(* PLC project Unnamed, Unknown Unnamed 1 *)
(* stored: creationDateTime 2022-08-16T15:49:17, modificationDateTime 2023-01-11T10:21:23 *)

PROGRAM Blink
  VAR
    blink_led AT %QX0.5 : BOOL;
  END_VAR
  VAR
    TON0 : TON;
    TOF0 : TOF;
  END_VAR

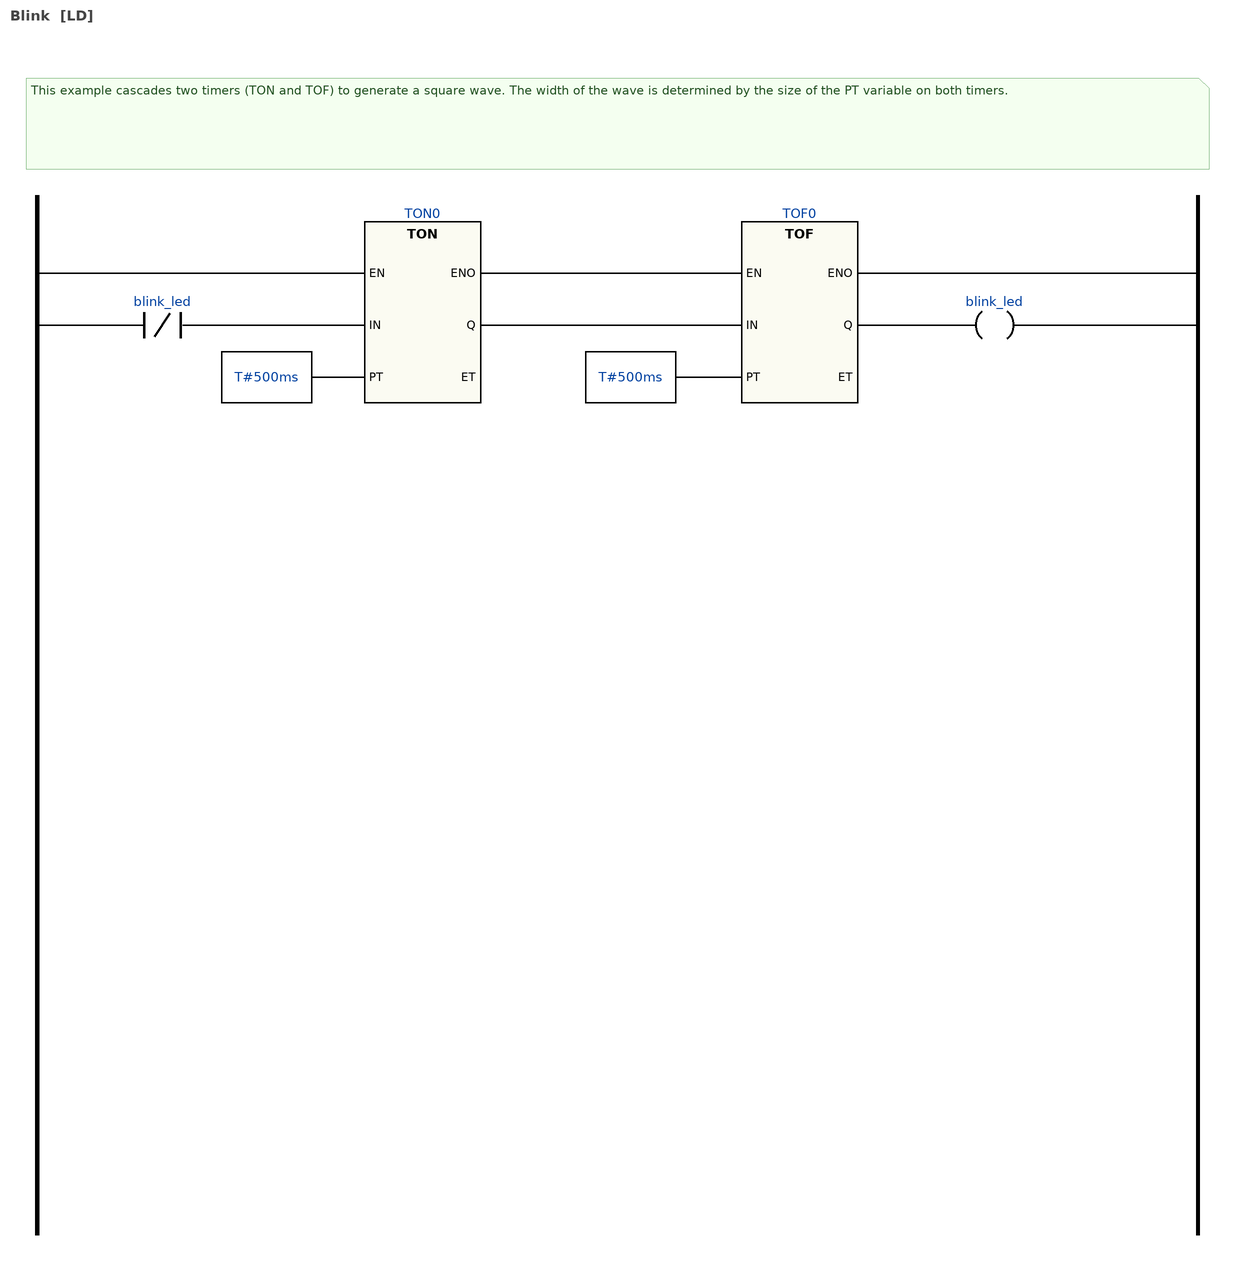
(* LD diagram, written out as Structured Text *)
(* This example cascades two timers (TON and TOF) to generate a square wave. The width of the wave is determined by the size of the PT variable on both timers. *)
TON0(IN := NOT blink_led, PT := T#500ms);
TOF0(EN := TON0.ENO, IN := TON0.Q, PT := T#500ms);
blink_led := TOF0.Q;
END_PROGRAM

CONFIGURATION Config0
  RESOURCE Res0 ON PLC
    TASK task0(INTERVAL := T#20ms, PRIORITY := 0);
    PROGRAM instance0 WITH task0 : Blink;
  END_RESOURCE
END_CONFIGURATION
